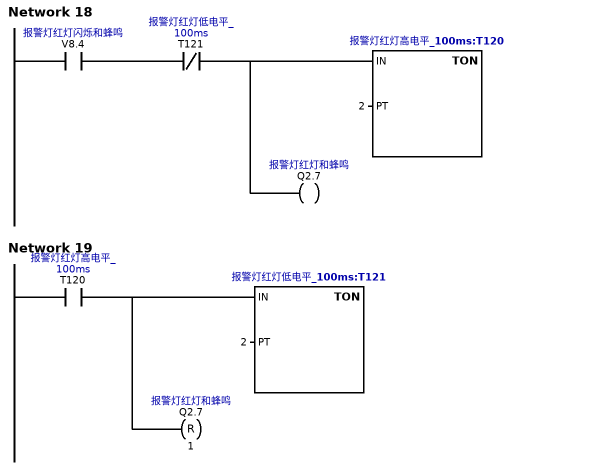
[picture p48: SBR21 networks 18-19]
Network 18
LD     报警灯红灯闪烁和蜂鸣:V8.4
AN     报警灯红灯低电平_100ms:T121
TON    报警灯红灯高电平_100ms:T120, 2
=      报警灯红灯和蜂鸣:Q2.7
Network 19
LD     报警灯红灯高电平_100ms:T120
TON    报警灯红灯低电平_100ms:T121, 2
R      报警灯红灯和蜂鸣:Q2.7, 1
END_SUBROUTINE_BLOCK
